(*********************************** G.D S.p.A. - Technical Department ***********************************
============= PROGRAM INFO ============
FOLDER:             TBD
MACHINES INVOLVED:  TBD 

============= DESCRIPTION =============
csp machine declaration

============= REVISIONS ===============
Date		Version	 	Author      	Description             
----------	-------		------------  	--------------------------------------------
2019/04/05 	0000.00	 	M.Grasso		Creation of the PRG

**********************************************************************************************************)
(*$R process_ref := prc; $*)
PROGRAM csp_case_feed_magazine_os
VAR
		
	prc:											process;
	prc_path:										STRING;
	
END_VAR

_read_var_input();

_object_manager();

IF NOT objects_running()
THEN
	RETURN;	
END_IF

_read_process_image();

_mode_manager();

_set_runtime_properties();

(********************************* BODY *********************************)
(************************************************************************)

_handle_messages();

_write_output();

ACTION _handle_messages:
;
END_ACTION

ACTION _handle_process_test:
;
END_ACTION

ACTION _mode_manager:
IF process_mode_req_is_pending(prc)
THEN
    process_apply_mode_req_first_step(prc);
    CASE process_get_mode(prc) OF
        MODE_TO_ABSENT:
			;
        MODE_TO_INACTIVE:
			;
        MODE_TO_TEST:
			;
        MODE_TO_OPERATIONAL:
			;
    END_CASE
    process_apply_mode_req_second_step(prc);
END_IF
END_ACTION

ACTION _object_manager:
IF objects_initialization()
THEN
	sub_process_init(
		object_name					:= 'csp_case_feed_magazine_os.prc', 
		process						:= csp_case_feed_magazine.prc, 
		CONVERSION_this				:= prc);
		
	prc_path 						:= process_get_path(prc);
END_IF

IF objects_running()
THEN
	process_cycle(prc);
END_IF
END_ACTION

ACTION _read_process_image:
;
END_ACTION

ACTION _read_var_input:
;
END_ACTION

ACTION _set_runtime_properties:
;
END_ACTION

ACTION _write_output:
;
END_ACTION

END_PROGRAM

(* stored: Version 1.1.0.1, ProductVersion 3.1.4022.12
   POU csp_case_feed_magazine_os: Id {563cb76d-b634-4271-8224-24cead4d19cd}, SpecialFunc None
   Action _handle_messages: Id {d92c0623-470e-4545-ad19-4de1420e9f0d}
   Action _handle_process_test: Id {b00e47f9-ab8b-46cb-9ed5-279d2122f682}
   Action _mode_manager: Id {b210b157-e57b-4b25-ac8f-dde9f2fa8cec}
   Action _object_manager: Id {314a6567-378d-46fc-be5b-30aa0c0784d9}
   Action _read_process_image: Id {7fdae3ee-8f9a-4261-875f-3a701149e756}
   Action _read_var_input: Id {ac90fd67-504a-4f96-a326-be60995ba615}
   Action _set_runtime_properties: Id {92d1ccb1-7c66-498e-b290-18a8b380e94a}
   Action _write_output: Id {51b45065-7887-4286-81b8-15868f03a824} *)
